PROGRAM MAIN
VAR
END_VAR

IF Allgemein.ImExport.bTriggerNewFileSelected THEN
	Allgemein.ImExport.bTriggerNewFileSelected := FALSE;
END_IF

IF Allgemein.ImExport.bTriggerNewFolderSelected THEN
	Allgemein.ImExport.bTriggerNewFolderSelected := FALSE;
END_IF

END_PROGRAM

(* stored: Version 1.1.0.1, ProductVersion 3.1.4024.4
   POU MAIN: Id {dbcb18db-7369-43c1-a98b-4ad572e1f264}, SpecialFunc None *)
